// TIA Portal V19 export
DATA_BLOCK "DI MAPING"   // DB1
{ S7_Optimized_Access := 'FALSE' }
   VAR
      "EMG STOP" : Bool;
      "HOOTER RESET_1" : Bool;
      "PHASE FAIL" : Bool;
      "AIR PRESSURE FAIL" : Bool;
      "SYRUP MFG VESSEL BOTTOM STERROR TRIP" : Bool;
      "PREMIXING VESSEL BOTTOM STERROR TRIP" : Bool;
      "INLINE 1 HOMOGENIZER MOTOR1 TRIP" : Bool;
      "INLINE 2 HOMOGENIZER MOTOR 2 TRIP" : Bool;
      "FILTER PRESS MOTOR 1 TRIP" : Bool;
      "FILTER PRESS MOTOR 2 TRIP" : Bool;
      "VACCUM PUMP MOTOR 1 TRIP" : Bool;
      "VACCUMP PUMP MOTOR 2 TRIP" : Bool;
      "VACCUMP PUMP MOTOR 3 TRIP" : Bool;
      "VACCUMP PUMP MOTOR 4 TRIP" : Bool;
      "SUGAR VESSEL BOTTOM STERROR TRIP" : Bool;
      "BASKET FILTER MOTOR TRIP" : Bool;
      "SYRUP FLOW SWITCH" : Bool;
      "PREMIXING FLOW SWITCH" : Bool;
      "SUGAR FLOW SWITCH" : Bool;
      "INLINE 1 FLOW SWITCH" : Bool;
      "INLINE 2 FLOW SWITCH" : Bool;
      "HOOTER RESET_2" : Bool;
      SPARE_DI1 : Bool;
      SPARE_DI2 : Bool;
      SPARE_DI3 : Bool;
      SPARE_DI4 : Bool;
      SPARE_DI5 : Bool;
      SPARE_DI6 : Bool;
      SPARE_DI7 : Bool;
      SPARE_DI8 : Bool;
      SPARE_DI9 : Bool;
      SPARE_DI10 : Bool;
   END_VAR
BEGIN
END_DATA_BLOCK
